// TIA Portal V20 export
TYPE "TypeCmd"
   STRUCT
      auto : Bool;   // automatic mode
      autoP : Bool;   // automatic plus
      autoM : Bool;   // automatic minus
      autoLift : Bool;   // automatic lift
      autoLower : Bool;   // automatic lower
      man : Bool;   // manual mode
      manP : Bool;   // manual plus
      manM : Bool;   // manual minus
      manLift : Bool;   // manual lift
      manLower : Bool;   // manual lower
      enable : Bool;   // release
      enPlus : Bool;   // release plus
      enMinus : Bool;   // release minus
      enLift : Bool;   // release lift
      enLower : Bool;   // release lower
      enAutoP : Bool;   // release automatic plus
      enAutoM : Bool;   // release automatic minus
      enAutoLift : Bool;   // release automatic lift
      enAutoLower : Bool;   // release automatic lower
      slow : Bool;
      lamp : Bool;   // indication lamp
      ack : Bool;   // fault acknowledge
      cycle : Bool;   // cycle start
      goToGpos : Bool;   // go to groundposition
      goToCpos : Bool;   // go to cm-position
      goToEpos : Bool;   // go to endpos
      goToWPos : Bool;   // go to wait/fly position
      inGpos : Bool;   // in groundposition
      inCpos : Bool;   // in cm-position
      inEpos : Bool;   // in endpos
      inWPos : Bool;   // in wait/fly position
      speed : Int;   // Desired speed raw in Hz or Upm
      tarSpeed : Real;   // target speed
      mmCycle : Real;   // milimeter per cycle
      gain : Real;   // gain
      ramp : Int;   // ramp
      startRamp : Int;   // start ramp
      stopRamp : Int;   // stop ramp
      gPos : Real;   // Desired value basic position [mm]
      cPos : Real;   // Desired value cm position [mm]
      ePos : Real;   // Desired value end position [mm]
      wPos : Real;   // Desired value wait/fly position [mm]
      tarMax : Real;   // target maximum
      tarMin : Real;   // target minimum
      target : Real;
      actual : Real;
   END_STRUCT;
END_TYPE
